// TIA Portal V19 export
FUNCTION_BLOCK "TYPIC_C701_IF_LBS"   // FB83, FBD
TITLE = TYPIC_C701_IF_LBS: Luchtbehandelingssysteem
{ S7_Optimized_Access := 'TRUE' }
AUTHOR : OCOTECH
FAMILY : Typical
NAME : C701.702
// Logisch Object Besturing: C701.702
// 
// De interne functie Luchtbehandelingssysteem verzorgt de interne besturing, bewaking en fysieke aansturing van de luchtgroep behorend tot de klimaatinstallatie.
// stored: MemoryReserve 10, SetENOAutomatically false
   VAR_INPUT
      STU_IF_LBS_CMD { ExternalAccessible := 'False'; ExternalVisible := 'False'; ExternalWritable := 'False'} : USInt;   // Sturing van de interne functie klimaatregeling (IF), luchtgroep
      IN_DME_PU { ExternalAccessible := 'False'; ExternalVisible := 'False'; ExternalWritable := 'False'} : Real;   // Drukmeting in pulsie kanaal
      IN_DME_EX { ExternalAccessible := 'False'; ExternalVisible := 'False'; ExternalWritable := 'False'} : Real;   // Drukmeting in extractie kanaal
      IN_TME_PU { ExternalAccessible := 'False'; ExternalVisible := 'False'; ExternalWritable := 'False'} : Real;   // Temperatuurmeting in pulsie kanaal
      IN_TME_EX { ExternalAccessible := 'False'; ExternalVisible := 'False'; ExternalWritable := 'False'} : Real;   // Temperatuurmeting in extractie kanaal
      IN_TME_BU { ExternalAccessible := 'False'; ExternalVisible := 'False'; ExternalWritable := 'False'} : Real;   // Temperatuurmeting buiten
      IN_VEN_PU { ExternalAccessible := 'False'; ExternalVisible := 'False'; ExternalWritable := 'False'} : Bool;   // Status pulsie ventilator (on/off)
      IN_VEN_PU_FB { ExternalAccessible := 'False'; ExternalVisible := 'False'; ExternalWritable := 'False'} : Real;   // Feedback snelheid pulsie ventilator
      IN_VEN_PU_AUT { ExternalAccessible := 'False'; ExternalVisible := 'False'; ExternalWritable := 'False'} : Bool;   // Status thermische beveiliging pulsie ventilator (1 = OK)
      IN_VEN_PU_SCW { ExternalAccessible := 'False'; ExternalVisible := 'False'; ExternalWritable := 'False'} : Bool;   // Werkschakelaar pulsie ventilator (1 = Aan)
      IN_VEN_EX { ExternalAccessible := 'False'; ExternalVisible := 'False'; ExternalWritable := 'False'} : Bool;   // Status extractie ventilator (on/off)
      IN_VEN_EX_FB { ExternalAccessible := 'False'; ExternalVisible := 'False'; ExternalWritable := 'False'} : Real;   // Feedback snelheid extractie ventilator
      IN_VEN_EX_AUT { ExternalAccessible := 'False'; ExternalVisible := 'False'; ExternalWritable := 'False'} : Bool;   // Status thermische beveiliging extractie ventilator (1 = OK)
      IN_VEN_EX_SCW { ExternalAccessible := 'False'; ExternalVisible := 'False'; ExternalWritable := 'False'} : Bool;   // Werkschakelaar extractie ventilator (1 = Aan)
      IN_KLR_KOB { ExternalAccessible := 'False'; ExternalVisible := 'False'; ExternalWritable := 'False'} : Real;   // Feedback stand 2weg klep koelbatterij
      IN_KLR_VEB { ExternalAccessible := 'False'; ExternalVisible := 'False'; ExternalWritable := 'False'} : Real;   // Feedback stand 3weg klep verwarmingsbatterij
      IN_KLR_PU { ExternalAccessible := 'False'; ExternalVisible := 'False'; ExternalWritable := 'False'} : Real;   // Terugmelding stand open/dicht register verse lucht
      IN_KLR_EX { ExternalAccessible := 'False'; ExternalVisible := 'False'; ExternalWritable := 'False'} : Real;   // Terugmelding stand open/dicht register extractie
      IN_KLR { ExternalAccessible := 'False'; ExternalVisible := 'False'; ExternalWritable := 'False'} : Real;   // Terugmelding stand mengregister
      IN_AVR { ExternalAccessible := 'False'; ExternalVisible := 'False'; ExternalWritable := 'False'} : Bool;   // Antivries schakelaar (1 = OK)
      IN_DME_FI_VL { ExternalAccessible := 'False'; ExternalVisible := 'False'; ExternalWritable := 'False'} : Bool;   // Drukverschilmeting filter verse lucht (1 = OK)
      IN_DME_FI_EX { ExternalAccessible := 'False'; ExternalVisible := 'False'; ExternalWritable := 'False'} : Bool;   // Drukverschilmeting filter extractie (1 = OK)
      IN_WMW { ExternalAccessible := 'False'; ExternalVisible := 'False'; ExternalWritable := 'False'} : Bool;   // Terugmelding status warmtewiel (Aan / Uit)
      IN_WMW_STO { ExternalAccessible := 'False'; ExternalVisible := 'False'; ExternalWritable := 'False'} : Bool;   // Fout warmtewiel (1 = OK)
      IN_BME { ExternalAccessible := 'False'; ExternalVisible := 'False'; ExternalWritable := 'False'} : Bool;   // Rookmelder (1 = OK)
      CFG_TYD_FB { ExternalAccessible := 'False'; ExternalVisible := 'False'; ExternalWritable := 'False'} : Time;   // Vertragingstijd storing foute terugmelding
   END_VAR
   VAR_OUTPUT
      VAR_IF_LBS { ExternalAccessible := 'False'; ExternalVisible := 'False'; ExternalWritable := 'False'} : "C701_VAR_IF_LBS_TYPIC";   // Struct met alle variabelen naar bovenliggende functies
      OUT_VEN_PU_VGV { ExternalAccessible := 'False'; ExternalVisible := 'False'; ExternalWritable := 'False'} : Bool;   // Vrijgave pulsie ventilator
      OUT_VEN_PU_SNE { ExternalAccessible := 'False'; ExternalVisible := 'False'; ExternalWritable := 'False'} : Real;   // Snelheid pulsie ventilator
      OUT_VEN_EX_VGV { ExternalAccessible := 'False'; ExternalVisible := 'False'; ExternalWritable := 'False'} : Bool;   // Vrijgave extractie ventilator
      OUT_VEN_EX_SNE { ExternalAccessible := 'False'; ExternalVisible := 'False'; ExternalWritable := 'False'} : Real;   // Snelheid extractie ventilator
      OUT_KLR_KOB { ExternalAccessible := 'False'; ExternalVisible := 'False'; ExternalWritable := 'False'} : Real;   // Aansturing klep koelbatterij
      OUT_KLR_VEB { ExternalAccessible := 'False'; ExternalVisible := 'False'; ExternalWritable := 'False'} : Real;   // Aansturing klep verwarmingsbatterij
      OUT_KLR_VL { ExternalAccessible := 'False'; ExternalVisible := 'False'; ExternalWritable := 'False'} : Real;   // Damper verse lucht sturing
      OUT_KLR_EX { ExternalAccessible := 'False'; ExternalVisible := 'False'; ExternalWritable := 'False'} : Real;   // Damper extractie lucht sturing
      OUT_KLR { ExternalAccessible := 'False'; ExternalVisible := 'False'; ExternalWritable := 'False'} : Real;   // Aansturing positie mengregister
      OUT_WMW { ExternalAccessible := 'False'; ExternalVisible := 'False'; ExternalWritable := 'False'} : Real;   // Aansturing recuperatie warmtewisselaar
   END_VAR
   VAR_IN_OUT
      STU_VGV_PMP_AAN : Bool;   // Vrijgave inschakelen
   END_VAR
   VAR
      BED : Struct   // Bedieningen
         REM : Bool;   // Bediening om luchtgroep in remote te schakelen
         NORMAAL : Bool;   // Bediening om luchtgroep in regime Normaal te schakelen
         RECIRCULATIE : Bool;   // Bediening om luchtgroep in regime Recirculatie te schakelen
         UIT : Bool;   // Bediening om luchtgroep in regime Uit te schakelen
      END_STRUCT;
      STO { ExternalWritable := 'False'} : Struct   // Storingen
         A001 : Bool;   // Storing van de motorbeveiliging van pulsie ventilator
         A002 : Bool;   // Storing van de motorbeveiliging van extractie ventilator
         A003 : Bool;   // Fout drukmeting pulsie
         A004 : Bool;   // Fout drukmeting extractie
         A005 : Bool;   // Fout temperatuurmeting pulsie
         A006 : Bool;   // Fout temperatuurmeting extractie
         A007 : Bool;   // Fout temperatuurmeting buitenlucht
         A008 : Bool;   // Antivries alarm
         A009 : Bool;   // Filter vuil verse lucht
         A010 : Bool;   // Filter vuil extractie lucht
         AT01 : Bool;   // Foute terugmelding: damper verse lucht aangestuurd, terugmelding niet (of te laat) ontvangen
         AT02 : Bool;   // Foute terugmelding: damper extractie lucht aangestuurd, terugmelding niet (of te laat) ontvangen
         M001 : Bool;   // De pulsie ventilator is afgekoppeld via de werkschakelaar
         M002 : Bool;   // De extractie ventilator is afgekoppeld via de werkschakelaar
      END_STRUCT;
      VAR { ExternalWritable := 'False'} : Struct   // Variabelen
         PID_P_PU : Real;   // P factor van PID regeling voor pulsie ventilator
         PID_I_PU : Time;   // Integratietijd van PID regeling voor pulsie ventilator
         PID_D_PU : Time;   // D actie van PID regeling voor pulsie ventilator
         PID_P_EX : Real;   // P factor van PID regeling voor extractie ventilator
         PID_I_EX : Time;   // Integratietijd van PID regeling voor extractie ventilator
         PID_D_EX : Time;   // D actie van PID regeling voor extractie ventilator
         PID_P_KOB : Real;   // P factor van PID regeling voor klep van koelbatterij
         PID_I_KOB : Time;   // Integratietijd van PID regeling voor klep van koelbatterij
         PID_D_KOB : Time;   // D actie van PID regeling voor klep van koelbatterij
         PID_P_VEB : Real;   // P factor van PID regeling voor klep van verwarmingsbatterij
         PID_I_VEB : Time;   // Integratietijd van PID regeling voor klep van verwarmingsbatterij
         PID_D_VEB : Time;   // D actie van PID regeling voor klep van verwarmingsbatterij
         SWA_D_PU : Real;   // Setpunt druk pulsie kanaal
         SWA_D_EX : Real;   // Setpunt druk extractie kanaal
         SWA_T_PU : Real;   // Setpunt temperatuur pulsie
         DME_PU : Real;   // Drukmeting pulsie kanaal
         DME_EX : Real;   // Drukmeting extractie kanaal
         TME_PU : Real;   // Temperatuurmeting in pulsie
         TME_EX : Real;   // Temperatuurmeting in extractie
         TME_BU : Real;   // Temperatuurmeting buitenlucht
         WRE { ExternalAccessible := 'False'; ExternalVisible := 'False'} : USInt;   // Werkingsregime
         BMO_HAND { ExternalAccessible := 'False'; ExternalVisible := 'False'} : Bool;   // TRUE = Werkingsregime is handmatig ingesteld via lokale bediening
         "Vrijgave pomp verwarmingsbat" { ExternalAccessible := 'False'; ExternalVisible := 'False'} : Bool;   // Gaat naar if verwarmingskring CHECKEN OF DEZE POMP NU HIER INZIT OF IN DE KRING
         REQ_VE { ExternalAccessible := 'False'; ExternalVisible := 'False'} : Bool;   // Warmtevraag voor kring verwarmingsbatterijen
         REQ_KO { ExternalAccessible := 'False'; ExternalVisible := 'False'} : Bool;   // Koelvraag voor kring koelbatterijen (luchtgroep)
      END_STRUCT;
   END_VAR
BEGIN

REGION Network 1: START
END_REGION

REGION Network 2: +++ Metingen +++
   // inlezen van de temperatuur en drukken.
END_REGION

REGION Network 3: +++ Storingen en meldingen +++
   // aanmaken van de storingen en meldingen.
END_REGION

REGION Network 4: Storing A001: Storing van de motorbeveiliging van pulsie ventilator
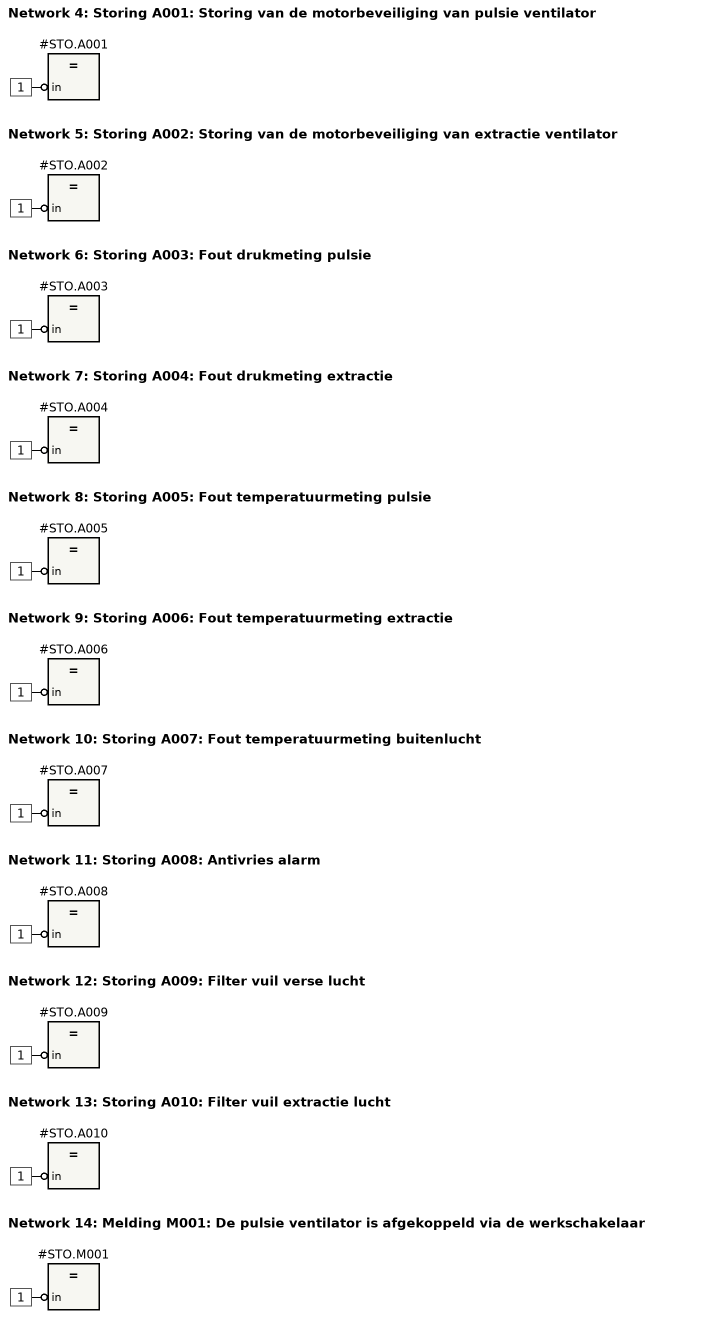
   #STO.A001 := NOT 1;
END_REGION

REGION Network 5: Storing A002: Storing van de motorbeveiliging van extractie ventilator
   #STO.A002 := NOT 1;
END_REGION

REGION Network 6: Storing A003: Fout drukmeting pulsie
   #STO.A003 := NOT 1;
END_REGION

REGION Network 7: Storing A004: Fout drukmeting extractie
   #STO.A004 := NOT 1;
END_REGION

REGION Network 8: Storing A005: Fout temperatuurmeting pulsie
   #STO.A005 := NOT 1;
END_REGION

REGION Network 9: Storing A006: Fout temperatuurmeting extractie
   #STO.A006 := NOT 1;
END_REGION

REGION Network 10: Storing A007: Fout temperatuurmeting buitenlucht
   #STO.A007 := NOT 1;
END_REGION

REGION Network 11: Storing A008: Antivries alarm
   #STO.A008 := NOT 1;
END_REGION

REGION Network 12: Storing A009: Filter vuil verse lucht
   #STO.A009 := NOT 1;
END_REGION

REGION Network 13: Storing A010: Filter vuil extractie lucht
   #STO.A010 := NOT 1;
END_REGION

REGION Network 14: Melding M001: De pulsie ventilator is afgekoppeld via de werkschakelaar
   #STO.M001 := NOT 1;
END_REGION

REGION Network 15: Melding M002: De extractie ventilator is afgekoppeld via de werkschakelaar
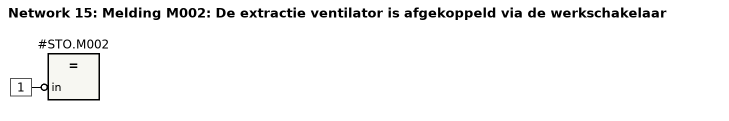
   #STO.M002 := NOT 1;
END_REGION

REGION Network 16: +++ Regelingen +++
   // PID regelingen voor luchtdebiet en temperatuur.
END_REGION

REGION Network 17: +++ Sturingen +++
   // aansturingen bepaalt door de uitgangen van de PID regelaars.
END_REGION

REGION Network 18 (SCL): EINDE
   // Variabelen van intern scada rakvlak naar outputs copieren
   #VAR_IF_LBS.WRE := #VAR.WRE;
   #VAR_IF_LBS.BMO_HAND := #VAR.BMO_HAND;
   #VAR_IF_LBS."Vrijgave pomp verwarmingsbat" := #VAR."Vrijgave pomp verwarmingsbat";
   #VAR_IF_LBS.REQ_VE := #VAR.REQ_VE;
   #VAR_IF_LBS.REQ_KO := #VAR.REQ_KO;
   #VAR_IF_LBS.STO := #STO;
END_REGION
END_FUNCTION_BLOCK
